// TIA Portal V20 export
TYPE "LER_typeBrakeTestEmControlNodes"
// stored: Access Published
   STRUCT
      commands { ExternalWritable := 'False'} : "LER_typeBrakeTestEmPlcCommands";
      monitoring { ExternalWritable := 'False'} : "LER_typeBrakeTestEmMonitoring";
   END_STRUCT;
END_TYPE
